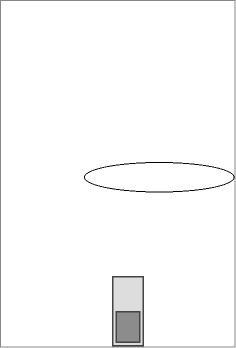
VISUALIZATION Visualization  // 236x348
    Ellipse (84,162 150x30)
    DipSwitch (93,276 70x70), variable: MAIN.bSignal, behaviour: TOGGLE, style: Switch-DipSwitch-Gray
END_VISUALIZATION

(* stored: Version 1.1.0.1, ProductVersion 3.1.4019.2
   Visu Visualization: Id {929de6f2-26a0-4cc0-acba-84afdd00a603} *)
